VISUALIZATION VISU_1  // 2x2
END_VISUALIZATION

(* stored: Version 1.1.0.1, ProductVersion 3.1.4022.18
   Visu VISU_1: Id {0cdb93bd-1d14-4b1a-9fb6-5da63c56ba02} *)
